// TIA Portal V16 export
// export: Created 2024-03-28T09:48:22.4867977Z, ExportSetting WithDefaults, DisplayName Totally Integrated Automation Portal, DisplayVersion V16, DisplayName TIA Portal Version Control Interface, DisplayVersion V16, DisplayName TIA Portal Openness, DisplayVersion V16, DisplayName STEP 7 Professional, DisplayVersion V16, DisplayName STEP 7 Safety, DisplayVersion V16, DisplayName WinCC Advanced, DisplayVersion V16
TYPE "UR_5_T2O_BitRegisters"
// stored: IsFailsafeCompliant false
   STRUCT
      Register : Array[0..63] of Bool;
   END_STRUCT;
END_TYPE
